/// machine data that is used through most sequences of the unit (motor speed, axes positions, ...)
TYPE PickerDataMachine :
STRUCT
  Slowspeed : LREAL;
  Highspeed : LREAL;
END_STRUCT
END_TYPE

(* stored: Version 1.1.0.1
   DUT PickerDataMachine: Id {9ada5900-7d28-4373-be9d-f14e4aa6e563} *)
